(* IEC 61131-3 sources: TIA2AX/tests/test_projects/expected/HW_2200220OffsetBodu_V18/A5, 6 files *)

(* ---- HwInputs.st ---- *)
TYPE
	HwInputs : STRUCT
		A6_15A2 AT %B0 : WORD;
		A6_15A3 AT %B2 : WORD;
		A6_15A4 AT %B4 : WORD;
		A6_15A9 AT %B6 : ARRAY[0..7] OF BYTE;
		_52K1_53AB1 AT %B157 : BYTE;
		_52K1_54AB2 AT %B158 : BYTE;
		_52K1_55AB3 AT %B159 : BYTE;
		_52K1_56AB4 AT %B160 : BYTE;
		_52K1_57AB5 AT %B179 : BYTE;
		_52K1_58AB6 AT %B147 : ARRAY[0..7] OF BYTE;
		_52K1_59AB7 AT %B45 : BYTE;
		_52K1_59aAB7 AT %B155 : BYTE;
		_52K1_60AB8 AT %B156 : BYTE;
		_52K1_61AB9 AT %B161 : BYTE;
		_52K1_62AB10 AT %B178 : BYTE;
		Bash_Input_1_byte_1 AT %B5300 : BYTE;
		Bash_Input_1_byte_2 AT %B5301 : BYTE;
		Bash_Input_2_word_1 AT %B5302 : DWORD;
		Bash_Input_1_word_1 AT %B5306 : WORD;
		Bash_Input_2_word_2 AT %B5308 : DWORD;
		Bash_Input_1_word_2 AT %B5312 : WORD;
		AEBDown_Input_1_byte_1 AT %B5314 : BYTE;
		AEBDown_Input_1_byte_2 AT %B5315 : BYTE;
		AEBDown_Input_2_word_1 AT %B5316 : DWORD;
		AEBDown_Input_1_word_1 AT %B5320 : WORD;
		AEBDown_Input_2_word_2 AT %B5322 : DWORD;
		AEBDown_Input_1_word_2 AT %B5326 : WORD;
		AEBUp_Input_1_byte_1 AT %B5328 : BYTE;
		AEBUp_Input_1_byte_2 AT %B5329 : BYTE;
		AEBUp_Input_2_word_1 AT %B5330 : DWORD;
		AEBUp_Input_1_word_1 AT %B5334 : WORD;
		AEBUp_Input_2_word_2 AT %B5336 : DWORD;
		AEBUp_Input_1_word_2 AT %B5340 : WORD;
		AETDown_Input_1_byte_1 AT %B5342 : BYTE;
		AETDown_Input_1_byte_2 AT %B5343 : BYTE;
		AETDown_Input_2_word_1 AT %B5344 : DWORD;
		AETDown_Input_1_word_1 AT %B5348 : WORD;
		AETDown_Input_2_word_2 AT %B5350 : DWORD;
		AETDown_Input_1_word_2 AT %B5354 : WORD;
		AETUp_Input_1_byte_1 AT %B5356 : BYTE;
		AETUp_Input_1_byte_2 AT %B5357 : BYTE;
		AETUp_Input_2_word_1 AT %B5358 : DWORD;
		AETUp_Input_1_word_1 AT %B5362 : WORD;
		AETUp_Input_2_word_2 AT %B5364 : DWORD;
		AETUp_Input_1_word_2 AT %B5368 : WORD;
		GT2_DL_PN1_1 AT %B162 : ARRAY[0..15] OF BYTE;
		GT2_B1 AT %B228 : ARRAY[0..6] OF BYTE;
		GT2_B2 AT %B221 : ARRAY[0..6] OF BYTE;
		GT2_B3 AT %B214 : ARRAY[0..6] OF BYTE;
		GT2_B4 AT %B207 : ARRAY[0..6] OF BYTE;
		GT2_B5 AT %B200 : ARRAY[0..6] OF BYTE;
		GT2_B6 AT %B189 : ARRAY[0..6] OF BYTE;
		GT2_B7 AT %B182 : ARRAY[0..6] OF BYTE;
		GT2_B8 AT %B235 : ARRAY[0..6] OF BYTE;
		GT2_B9 AT %B242 : ARRAY[0..6] OF BYTE;
		CPX_CW_SW AT %B71 : DWORD;
		CPX_CNC AT %B408 : ARRAY[0..31] OF BYTE;
		CPX_PtP AT %B385 : ARRAY[0..15] OF BYTE;
		CPX_Error AT %B440 : ARRAY[0..31] OF BYTE;
		Reader_Handshake_and_General_Error_Status_Bits_1 AT %B15 : BYTE;
		Reader_BUSY_Status_Bits_1 AT %B16 : BYTE;
		Reader_Completion_Status_Bits_1 AT %B17 : BYTE;
		Reader_Error_Status_Bits_1 AT %B18 : BYTE;
		Reader_Terminal_Status_Bits_1 AT %B19 : BYTE;
		Reader_Unstable_Read_Status_Bits_1 AT %B20 : BYTE;
		Reader_Matching_Level_and_Total_Evaluation_Grade_Status_1 AT %B21 : ARRAY[0..7] OF BYTE;
		Reader_Operation_Result_Status_1 AT %B51 : ARRAY[0..19] OF BYTE;
		Reader_Read_Data_128Byte_1 AT %B249 : ARRAY[0..135] OF BYTE;
	END_STRUCT;
END_TYPE

(* ---- HwOutputs.st ---- *)
TYPE
	HwOutputs : STRUCT
		A6_15A5 AT %B1 : WORD;
		A6_15A6 AT %B3 : WORD;
		A6_15A7 AT %B14 : WORD;
		A6_15A8 AT %B16 : WORD;
		A6_15A10 AT %B99 : ARRAY[0..7] OF BYTE;
		VI_13_MPA1S_VMPA1_FB_EMS_8_8DO_1 AT %B6 : BYTE;
		VI_13_MPA1S_VMPA1_FB_EMS_8_8DO_2 AT %B8 : BYTE;
		VI_13_MPA1S_VMPA1_FB_EMS_8_8DO_3 AT %B9 : BYTE;
		VI_13_MPA1S_VMPA1_FB_EMS_8_8DO_4 AT %B10 : BYTE;
		VI_13_MPA1S_VMPA1_FB_EMS_8_8DO_5 AT %B11 : BYTE;
		VI_13_MPA1S_VMPA1_FB_EMS_8_8DO_6 AT %B12 : BYTE;
		VI_13_MPA1S_VMPA1_FB_EMS_8_8DO_7 AT %B13 : BYTE;
		VI_13_MPA1S_VMPA1_FB_EMS_8_8DO_8 AT %B18 : BYTE;
		Bash_Output_1_byte_1 AT %B5300 : BYTE;
		Bash_Output_1_byte_2 AT %B5301 : BYTE;
		AEBDown_Output_1_byte_1 AT %B5302 : BYTE;
		AEBDown_Output_1_byte_2 AT %B5303 : BYTE;
		AEBUp_Output_1_byte_1 AT %B5304 : BYTE;
		AEBUp_Output_1_byte_2 AT %B5305 : BYTE;
		AETDown_Output_1_byte_1 AT %B5306 : BYTE;
		AETDown_Output_1_byte_2 AT %B5307 : BYTE;
		AETUp_Output_1_byte_1 AT %B5308 : BYTE;
		AETUp_Output_1_byte_2 AT %B5309 : BYTE;
		GT2_DL_PN1_1 AT %B32 : BYTE;
		GT2_B1 AT %B45 : BYTE;
		GT2_B2 AT %B147 : BYTE;
		GT2_B3 AT %B148 : BYTE;
		GT2_B4 AT %B149 : BYTE;
		GT2_B5 AT %B39 : BYTE;
		GT2_B6 AT %B38 : BYTE;
		GT2_B7 AT %B150 : BYTE;
		GT2_B8 AT %B151 : BYTE;
		GT2_B9 AT %B33 : BYTE;
		CPX_CW_SW AT %B21 : DWORD;
		CPX_CNC AT %B51 : ARRAY[0..31] OF BYTE;
		CPX_PtP AT %B83 : ARRAY[0..15] OF BYTE;
		CPX_Error AT %B282 : ARRAY[0..31] OF BYTE;
		Reader_Latch_and_Error_Clear_Control_Bits_1 AT %B0 : BYTE;
		Reader_Operation_instruction_Control_Bits_1 AT %B5 : BYTE;
		Reader_Completion_Clear_Control_Bits_1 AT %B7 : BYTE;
		Reader_Parameter_Bank_Number_1 AT %B19 : WORD;
		Reader_User_Data_128Byte_1 AT %B152 : ARRAY[0..129] OF BYTE;
	END_STRUCT;
END_TYPE

(* ---- PlcInputs.st ---- *)
TYPE
	PlcInputs : STRUCT
		A6_15A2 : WORD;
		A6_15A3 : WORD;
		A6_15A4 : WORD;
		A6_15A9 : ARRAY[0..7] OF BYTE;
		_52K1_53AB1 : BYTE;
		_52K1_54AB2 : BYTE;
		_52K1_55AB3 : BYTE;
		_52K1_56AB4 : BYTE;
		_52K1_57AB5 : BYTE;
		_52K1_58AB6 : ARRAY[0..7] OF BYTE;
		_52K1_59AB7 : BYTE;
		_52K1_59aAB7 : BYTE;
		_52K1_60AB8 : BYTE;
		_52K1_61AB9 : BYTE;
		_52K1_62AB10 : BYTE;
		Bash_Input_1_byte_1 : BYTE;
		Bash_Input_1_byte_2 : BYTE;
		Bash_Input_2_word_1 : DWORD;
		Bash_Input_1_word_1 : WORD;
		Bash_Input_2_word_2 : DWORD;
		Bash_Input_1_word_2 : WORD;
		AEBDown_Input_1_byte_1 : BYTE;
		AEBDown_Input_1_byte_2 : BYTE;
		AEBDown_Input_2_word_1 : DWORD;
		AEBDown_Input_1_word_1 : WORD;
		AEBDown_Input_2_word_2 : DWORD;
		AEBDown_Input_1_word_2 : WORD;
		AEBUp_Input_1_byte_1 : BYTE;
		AEBUp_Input_1_byte_2 : BYTE;
		AEBUp_Input_2_word_1 : DWORD;
		AEBUp_Input_1_word_1 : WORD;
		AEBUp_Input_2_word_2 : DWORD;
		AEBUp_Input_1_word_2 : WORD;
		AETDown_Input_1_byte_1 : BYTE;
		AETDown_Input_1_byte_2 : BYTE;
		AETDown_Input_2_word_1 : DWORD;
		AETDown_Input_1_word_1 : WORD;
		AETDown_Input_2_word_2 : DWORD;
		AETDown_Input_1_word_2 : WORD;
		AETUp_Input_1_byte_1 : BYTE;
		AETUp_Input_1_byte_2 : BYTE;
		AETUp_Input_2_word_1 : DWORD;
		AETUp_Input_1_word_1 : WORD;
		AETUp_Input_2_word_2 : DWORD;
		AETUp_Input_1_word_2 : WORD;
		GT2_DL_PN1_1 : ARRAY[0..15] OF BYTE;
		GT2_B1 : ARRAY[0..6] OF BYTE;
		GT2_B2 : ARRAY[0..6] OF BYTE;
		GT2_B3 : ARRAY[0..6] OF BYTE;
		GT2_B4 : ARRAY[0..6] OF BYTE;
		GT2_B5 : ARRAY[0..6] OF BYTE;
		GT2_B6 : ARRAY[0..6] OF BYTE;
		GT2_B7 : ARRAY[0..6] OF BYTE;
		GT2_B8 : ARRAY[0..6] OF BYTE;
		GT2_B9 : ARRAY[0..6] OF BYTE;
		CPX_CW_SW : DWORD;
		CPX_CNC : ARRAY[0..31] OF BYTE;
		CPX_PtP : ARRAY[0..15] OF BYTE;
		CPX_Error : ARRAY[0..31] OF BYTE;
		Reader_Handshake_and_General_Error_Status_Bits_1 : BYTE;
		Reader_BUSY_Status_Bits_1 : BYTE;
		Reader_Completion_Status_Bits_1 : BYTE;
		Reader_Error_Status_Bits_1 : BYTE;
		Reader_Terminal_Status_Bits_1 : BYTE;
		Reader_Unstable_Read_Status_Bits_1 : BYTE;
		Reader_Matching_Level_and_Total_Evaluation_Grade_Status_1 : ARRAY[0..7] OF BYTE;
		Reader_Operation_Result_Status_1 : ARRAY[0..19] OF BYTE;
		Reader_Read_Data_128Byte_1 : ARRAY[0..135] OF BYTE;
	END_STRUCT;
END_TYPE

(* ---- PlcOutputs.st ---- *)
TYPE
	PlcOutputs : STRUCT
		A6_15A5 : WORD;
		A6_15A6 : WORD;
		A6_15A7 : WORD;
		A6_15A8 : WORD;
		A6_15A10 : ARRAY[0..7] OF BYTE;
		VI_13_MPA1S_VMPA1_FB_EMS_8_8DO_1 : BYTE;
		VI_13_MPA1S_VMPA1_FB_EMS_8_8DO_2 : BYTE;
		VI_13_MPA1S_VMPA1_FB_EMS_8_8DO_3 : BYTE;
		VI_13_MPA1S_VMPA1_FB_EMS_8_8DO_4 : BYTE;
		VI_13_MPA1S_VMPA1_FB_EMS_8_8DO_5 : BYTE;
		VI_13_MPA1S_VMPA1_FB_EMS_8_8DO_6 : BYTE;
		VI_13_MPA1S_VMPA1_FB_EMS_8_8DO_7 : BYTE;
		VI_13_MPA1S_VMPA1_FB_EMS_8_8DO_8 : BYTE;
		Bash_Output_1_byte_1 : BYTE;
		Bash_Output_1_byte_2 : BYTE;
		AEBDown_Output_1_byte_1 : BYTE;
		AEBDown_Output_1_byte_2 : BYTE;
		AEBUp_Output_1_byte_1 : BYTE;
		AEBUp_Output_1_byte_2 : BYTE;
		AETDown_Output_1_byte_1 : BYTE;
		AETDown_Output_1_byte_2 : BYTE;
		AETUp_Output_1_byte_1 : BYTE;
		AETUp_Output_1_byte_2 : BYTE;
		GT2_DL_PN1_1 : BYTE;
		GT2_B1 : BYTE;
		GT2_B2 : BYTE;
		GT2_B3 : BYTE;
		GT2_B4 : BYTE;
		GT2_B5 : BYTE;
		GT2_B6 : BYTE;
		GT2_B7 : BYTE;
		GT2_B8 : BYTE;
		GT2_B9 : BYTE;
		CPX_CW_SW : DWORD;
		CPX_CNC : ARRAY[0..31] OF BYTE;
		CPX_PtP : ARRAY[0..15] OF BYTE;
		CPX_Error : ARRAY[0..31] OF BYTE;
		Reader_Latch_and_Error_Clear_Control_Bits_1 : BYTE;
		Reader_Operation_instruction_Control_Bits_1 : BYTE;
		Reader_Completion_Clear_Control_Bits_1 : BYTE;
		Reader_Parameter_Bank_Number_1 : WORD;
		Reader_User_Data_128Byte_1 : ARRAY[0..129] OF BYTE;
	END_STRUCT;
END_TYPE

(* ---- CopyInputs.st ---- *)
FUNCTION CopyInputs
	VAR_EXTERNAL
		HwInputs : HwInputs;
		PlcInputs : PlcInputs;
	END_VAR
	PlcInputs.A6_15A2 := HwInputs.A6_15A2;
	PlcInputs.A6_15A3 := HwInputs.A6_15A3;
	PlcInputs.A6_15A4 := HwInputs.A6_15A4;
	PlcInputs.A6_15A9[0] := HwInputs.A6_15A9[0];
	PlcInputs.A6_15A9[1] := HwInputs.A6_15A9[1];
	PlcInputs.A6_15A9[2] := HwInputs.A6_15A9[2];
	PlcInputs.A6_15A9[3] := HwInputs.A6_15A9[3];
	PlcInputs.A6_15A9[4] := HwInputs.A6_15A9[4];
	PlcInputs.A6_15A9[5] := HwInputs.A6_15A9[5];
	PlcInputs.A6_15A9[6] := HwInputs.A6_15A9[6];
	PlcInputs.A6_15A9[7] := HwInputs.A6_15A9[7];
	PlcInputs._52K1_53AB1 := HwInputs._52K1_53AB1;
	PlcInputs._52K1_54AB2 := HwInputs._52K1_54AB2;
	PlcInputs._52K1_55AB3 := HwInputs._52K1_55AB3;
	PlcInputs._52K1_56AB4 := HwInputs._52K1_56AB4;
	PlcInputs._52K1_57AB5 := HwInputs._52K1_57AB5;
	PlcInputs._52K1_58AB6[0] := HwInputs._52K1_58AB6[0];
	PlcInputs._52K1_58AB6[1] := HwInputs._52K1_58AB6[1];
	PlcInputs._52K1_58AB6[2] := HwInputs._52K1_58AB6[2];
	PlcInputs._52K1_58AB6[3] := HwInputs._52K1_58AB6[3];
	PlcInputs._52K1_58AB6[4] := HwInputs._52K1_58AB6[4];
	PlcInputs._52K1_58AB6[5] := HwInputs._52K1_58AB6[5];
	PlcInputs._52K1_58AB6[6] := HwInputs._52K1_58AB6[6];
	PlcInputs._52K1_58AB6[7] := HwInputs._52K1_58AB6[7];
	PlcInputs._52K1_59AB7 := HwInputs._52K1_59AB7;
	PlcInputs._52K1_59aAB7 := HwInputs._52K1_59aAB7;
	PlcInputs._52K1_60AB8 := HwInputs._52K1_60AB8;
	PlcInputs._52K1_61AB9 := HwInputs._52K1_61AB9;
	PlcInputs._52K1_62AB10 := HwInputs._52K1_62AB10;
	PlcInputs.Bash_Input_1_byte_1 := HwInputs.Bash_Input_1_byte_1;
	PlcInputs.Bash_Input_1_byte_2 := HwInputs.Bash_Input_1_byte_2;
	PlcInputs.Bash_Input_2_word_1 := HwInputs.Bash_Input_2_word_1;
	PlcInputs.Bash_Input_1_word_1 := HwInputs.Bash_Input_1_word_1;
	PlcInputs.Bash_Input_2_word_2 := HwInputs.Bash_Input_2_word_2;
	PlcInputs.Bash_Input_1_word_2 := HwInputs.Bash_Input_1_word_2;
	PlcInputs.AEBDown_Input_1_byte_1 := HwInputs.AEBDown_Input_1_byte_1;
	PlcInputs.AEBDown_Input_1_byte_2 := HwInputs.AEBDown_Input_1_byte_2;
	PlcInputs.AEBDown_Input_2_word_1 := HwInputs.AEBDown_Input_2_word_1;
	PlcInputs.AEBDown_Input_1_word_1 := HwInputs.AEBDown_Input_1_word_1;
	PlcInputs.AEBDown_Input_2_word_2 := HwInputs.AEBDown_Input_2_word_2;
	PlcInputs.AEBDown_Input_1_word_2 := HwInputs.AEBDown_Input_1_word_2;
	PlcInputs.AEBUp_Input_1_byte_1 := HwInputs.AEBUp_Input_1_byte_1;
	PlcInputs.AEBUp_Input_1_byte_2 := HwInputs.AEBUp_Input_1_byte_2;
	PlcInputs.AEBUp_Input_2_word_1 := HwInputs.AEBUp_Input_2_word_1;
	PlcInputs.AEBUp_Input_1_word_1 := HwInputs.AEBUp_Input_1_word_1;
	PlcInputs.AEBUp_Input_2_word_2 := HwInputs.AEBUp_Input_2_word_2;
	PlcInputs.AEBUp_Input_1_word_2 := HwInputs.AEBUp_Input_1_word_2;
	PlcInputs.AETDown_Input_1_byte_1 := HwInputs.AETDown_Input_1_byte_1;
	PlcInputs.AETDown_Input_1_byte_2 := HwInputs.AETDown_Input_1_byte_2;
	PlcInputs.AETDown_Input_2_word_1 := HwInputs.AETDown_Input_2_word_1;
	PlcInputs.AETDown_Input_1_word_1 := HwInputs.AETDown_Input_1_word_1;
	PlcInputs.AETDown_Input_2_word_2 := HwInputs.AETDown_Input_2_word_2;
	PlcInputs.AETDown_Input_1_word_2 := HwInputs.AETDown_Input_1_word_2;
	PlcInputs.AETUp_Input_1_byte_1 := HwInputs.AETUp_Input_1_byte_1;
	PlcInputs.AETUp_Input_1_byte_2 := HwInputs.AETUp_Input_1_byte_2;
	PlcInputs.AETUp_Input_2_word_1 := HwInputs.AETUp_Input_2_word_1;
	PlcInputs.AETUp_Input_1_word_1 := HwInputs.AETUp_Input_1_word_1;
	PlcInputs.AETUp_Input_2_word_2 := HwInputs.AETUp_Input_2_word_2;
	PlcInputs.AETUp_Input_1_word_2 := HwInputs.AETUp_Input_1_word_2;
	PlcInputs.GT2_DL_PN1_1[0] := HwInputs.GT2_DL_PN1_1[0];
	PlcInputs.GT2_DL_PN1_1[1] := HwInputs.GT2_DL_PN1_1[1];
	PlcInputs.GT2_DL_PN1_1[2] := HwInputs.GT2_DL_PN1_1[2];
	PlcInputs.GT2_DL_PN1_1[3] := HwInputs.GT2_DL_PN1_1[3];
	PlcInputs.GT2_DL_PN1_1[4] := HwInputs.GT2_DL_PN1_1[4];
	PlcInputs.GT2_DL_PN1_1[5] := HwInputs.GT2_DL_PN1_1[5];
	PlcInputs.GT2_DL_PN1_1[6] := HwInputs.GT2_DL_PN1_1[6];
	PlcInputs.GT2_DL_PN1_1[7] := HwInputs.GT2_DL_PN1_1[7];
	PlcInputs.GT2_DL_PN1_1[8] := HwInputs.GT2_DL_PN1_1[8];
	PlcInputs.GT2_DL_PN1_1[9] := HwInputs.GT2_DL_PN1_1[9];
	PlcInputs.GT2_DL_PN1_1[10] := HwInputs.GT2_DL_PN1_1[10];
	PlcInputs.GT2_DL_PN1_1[11] := HwInputs.GT2_DL_PN1_1[11];
	PlcInputs.GT2_DL_PN1_1[12] := HwInputs.GT2_DL_PN1_1[12];
	PlcInputs.GT2_DL_PN1_1[13] := HwInputs.GT2_DL_PN1_1[13];
	PlcInputs.GT2_DL_PN1_1[14] := HwInputs.GT2_DL_PN1_1[14];
	PlcInputs.GT2_DL_PN1_1[15] := HwInputs.GT2_DL_PN1_1[15];
	PlcInputs.GT2_B1[0] := HwInputs.GT2_B1[0];
	PlcInputs.GT2_B1[1] := HwInputs.GT2_B1[1];
	PlcInputs.GT2_B1[2] := HwInputs.GT2_B1[2];
	PlcInputs.GT2_B1[3] := HwInputs.GT2_B1[3];
	PlcInputs.GT2_B1[4] := HwInputs.GT2_B1[4];
	PlcInputs.GT2_B1[5] := HwInputs.GT2_B1[5];
	PlcInputs.GT2_B1[6] := HwInputs.GT2_B1[6];
	PlcInputs.GT2_B2[0] := HwInputs.GT2_B2[0];
	PlcInputs.GT2_B2[1] := HwInputs.GT2_B2[1];
	PlcInputs.GT2_B2[2] := HwInputs.GT2_B2[2];
	PlcInputs.GT2_B2[3] := HwInputs.GT2_B2[3];
	PlcInputs.GT2_B2[4] := HwInputs.GT2_B2[4];
	PlcInputs.GT2_B2[5] := HwInputs.GT2_B2[5];
	PlcInputs.GT2_B2[6] := HwInputs.GT2_B2[6];
	PlcInputs.GT2_B3[0] := HwInputs.GT2_B3[0];
	PlcInputs.GT2_B3[1] := HwInputs.GT2_B3[1];
	PlcInputs.GT2_B3[2] := HwInputs.GT2_B3[2];
	PlcInputs.GT2_B3[3] := HwInputs.GT2_B3[3];
	PlcInputs.GT2_B3[4] := HwInputs.GT2_B3[4];
	PlcInputs.GT2_B3[5] := HwInputs.GT2_B3[5];
	PlcInputs.GT2_B3[6] := HwInputs.GT2_B3[6];
	PlcInputs.GT2_B4[0] := HwInputs.GT2_B4[0];
	PlcInputs.GT2_B4[1] := HwInputs.GT2_B4[1];
	PlcInputs.GT2_B4[2] := HwInputs.GT2_B4[2];
	PlcInputs.GT2_B4[3] := HwInputs.GT2_B4[3];
	PlcInputs.GT2_B4[4] := HwInputs.GT2_B4[4];
	PlcInputs.GT2_B4[5] := HwInputs.GT2_B4[5];
	PlcInputs.GT2_B4[6] := HwInputs.GT2_B4[6];
	PlcInputs.GT2_B5[0] := HwInputs.GT2_B5[0];
	PlcInputs.GT2_B5[1] := HwInputs.GT2_B5[1];
	PlcInputs.GT2_B5[2] := HwInputs.GT2_B5[2];
	PlcInputs.GT2_B5[3] := HwInputs.GT2_B5[3];
	PlcInputs.GT2_B5[4] := HwInputs.GT2_B5[4];
	PlcInputs.GT2_B5[5] := HwInputs.GT2_B5[5];
	PlcInputs.GT2_B5[6] := HwInputs.GT2_B5[6];
	PlcInputs.GT2_B6[0] := HwInputs.GT2_B6[0];
	PlcInputs.GT2_B6[1] := HwInputs.GT2_B6[1];
	PlcInputs.GT2_B6[2] := HwInputs.GT2_B6[2];
	PlcInputs.GT2_B6[3] := HwInputs.GT2_B6[3];
	PlcInputs.GT2_B6[4] := HwInputs.GT2_B6[4];
	PlcInputs.GT2_B6[5] := HwInputs.GT2_B6[5];
	PlcInputs.GT2_B6[6] := HwInputs.GT2_B6[6];
	PlcInputs.GT2_B7[0] := HwInputs.GT2_B7[0];
	PlcInputs.GT2_B7[1] := HwInputs.GT2_B7[1];
	PlcInputs.GT2_B7[2] := HwInputs.GT2_B7[2];
	PlcInputs.GT2_B7[3] := HwInputs.GT2_B7[3];
	PlcInputs.GT2_B7[4] := HwInputs.GT2_B7[4];
	PlcInputs.GT2_B7[5] := HwInputs.GT2_B7[5];
	PlcInputs.GT2_B7[6] := HwInputs.GT2_B7[6];
	PlcInputs.GT2_B8[0] := HwInputs.GT2_B8[0];
	PlcInputs.GT2_B8[1] := HwInputs.GT2_B8[1];
	PlcInputs.GT2_B8[2] := HwInputs.GT2_B8[2];
	PlcInputs.GT2_B8[3] := HwInputs.GT2_B8[3];
	PlcInputs.GT2_B8[4] := HwInputs.GT2_B8[4];
	PlcInputs.GT2_B8[5] := HwInputs.GT2_B8[5];
	PlcInputs.GT2_B8[6] := HwInputs.GT2_B8[6];
	PlcInputs.GT2_B9[0] := HwInputs.GT2_B9[0];
	PlcInputs.GT2_B9[1] := HwInputs.GT2_B9[1];
	PlcInputs.GT2_B9[2] := HwInputs.GT2_B9[2];
	PlcInputs.GT2_B9[3] := HwInputs.GT2_B9[3];
	PlcInputs.GT2_B9[4] := HwInputs.GT2_B9[4];
	PlcInputs.GT2_B9[5] := HwInputs.GT2_B9[5];
	PlcInputs.GT2_B9[6] := HwInputs.GT2_B9[6];
	PlcInputs.CPX_CW_SW := HwInputs.CPX_CW_SW;
	PlcInputs.CPX_CNC[0] := HwInputs.CPX_CNC[0];
	PlcInputs.CPX_CNC[1] := HwInputs.CPX_CNC[1];
	PlcInputs.CPX_CNC[2] := HwInputs.CPX_CNC[2];
	PlcInputs.CPX_CNC[3] := HwInputs.CPX_CNC[3];
	PlcInputs.CPX_CNC[4] := HwInputs.CPX_CNC[4];
	PlcInputs.CPX_CNC[5] := HwInputs.CPX_CNC[5];
	PlcInputs.CPX_CNC[6] := HwInputs.CPX_CNC[6];
	PlcInputs.CPX_CNC[7] := HwInputs.CPX_CNC[7];
	PlcInputs.CPX_CNC[8] := HwInputs.CPX_CNC[8];
	PlcInputs.CPX_CNC[9] := HwInputs.CPX_CNC[9];
	PlcInputs.CPX_CNC[10] := HwInputs.CPX_CNC[10];
	PlcInputs.CPX_CNC[11] := HwInputs.CPX_CNC[11];
	PlcInputs.CPX_CNC[12] := HwInputs.CPX_CNC[12];
	PlcInputs.CPX_CNC[13] := HwInputs.CPX_CNC[13];
	PlcInputs.CPX_CNC[14] := HwInputs.CPX_CNC[14];
	PlcInputs.CPX_CNC[15] := HwInputs.CPX_CNC[15];
	PlcInputs.CPX_CNC[16] := HwInputs.CPX_CNC[16];
	PlcInputs.CPX_CNC[17] := HwInputs.CPX_CNC[17];
	PlcInputs.CPX_CNC[18] := HwInputs.CPX_CNC[18];
	PlcInputs.CPX_CNC[19] := HwInputs.CPX_CNC[19];
	PlcInputs.CPX_CNC[20] := HwInputs.CPX_CNC[20];
	PlcInputs.CPX_CNC[21] := HwInputs.CPX_CNC[21];
	PlcInputs.CPX_CNC[22] := HwInputs.CPX_CNC[22];
	PlcInputs.CPX_CNC[23] := HwInputs.CPX_CNC[23];
	PlcInputs.CPX_CNC[24] := HwInputs.CPX_CNC[24];
	PlcInputs.CPX_CNC[25] := HwInputs.CPX_CNC[25];
	PlcInputs.CPX_CNC[26] := HwInputs.CPX_CNC[26];
	PlcInputs.CPX_CNC[27] := HwInputs.CPX_CNC[27];
	PlcInputs.CPX_CNC[28] := HwInputs.CPX_CNC[28];
	PlcInputs.CPX_CNC[29] := HwInputs.CPX_CNC[29];
	PlcInputs.CPX_CNC[30] := HwInputs.CPX_CNC[30];
	PlcInputs.CPX_CNC[31] := HwInputs.CPX_CNC[31];
	PlcInputs.CPX_PtP[0] := HwInputs.CPX_PtP[0];
	PlcInputs.CPX_PtP[1] := HwInputs.CPX_PtP[1];
	PlcInputs.CPX_PtP[2] := HwInputs.CPX_PtP[2];
	PlcInputs.CPX_PtP[3] := HwInputs.CPX_PtP[3];
	PlcInputs.CPX_PtP[4] := HwInputs.CPX_PtP[4];
	PlcInputs.CPX_PtP[5] := HwInputs.CPX_PtP[5];
	PlcInputs.CPX_PtP[6] := HwInputs.CPX_PtP[6];
	PlcInputs.CPX_PtP[7] := HwInputs.CPX_PtP[7];
	PlcInputs.CPX_PtP[8] := HwInputs.CPX_PtP[8];
	PlcInputs.CPX_PtP[9] := HwInputs.CPX_PtP[9];
	PlcInputs.CPX_PtP[10] := HwInputs.CPX_PtP[10];
	PlcInputs.CPX_PtP[11] := HwInputs.CPX_PtP[11];
	PlcInputs.CPX_PtP[12] := HwInputs.CPX_PtP[12];
	PlcInputs.CPX_PtP[13] := HwInputs.CPX_PtP[13];
	PlcInputs.CPX_PtP[14] := HwInputs.CPX_PtP[14];
	PlcInputs.CPX_PtP[15] := HwInputs.CPX_PtP[15];
	PlcInputs.CPX_Error[0] := HwInputs.CPX_Error[0];
	PlcInputs.CPX_Error[1] := HwInputs.CPX_Error[1];
	PlcInputs.CPX_Error[2] := HwInputs.CPX_Error[2];
	PlcInputs.CPX_Error[3] := HwInputs.CPX_Error[3];
	PlcInputs.CPX_Error[4] := HwInputs.CPX_Error[4];
	PlcInputs.CPX_Error[5] := HwInputs.CPX_Error[5];
	PlcInputs.CPX_Error[6] := HwInputs.CPX_Error[6];
	PlcInputs.CPX_Error[7] := HwInputs.CPX_Error[7];
	PlcInputs.CPX_Error[8] := HwInputs.CPX_Error[8];
	PlcInputs.CPX_Error[9] := HwInputs.CPX_Error[9];
	PlcInputs.CPX_Error[10] := HwInputs.CPX_Error[10];
	PlcInputs.CPX_Error[11] := HwInputs.CPX_Error[11];
	PlcInputs.CPX_Error[12] := HwInputs.CPX_Error[12];
	PlcInputs.CPX_Error[13] := HwInputs.CPX_Error[13];
	PlcInputs.CPX_Error[14] := HwInputs.CPX_Error[14];
	PlcInputs.CPX_Error[15] := HwInputs.CPX_Error[15];
	PlcInputs.CPX_Error[16] := HwInputs.CPX_Error[16];
	PlcInputs.CPX_Error[17] := HwInputs.CPX_Error[17];
	PlcInputs.CPX_Error[18] := HwInputs.CPX_Error[18];
	PlcInputs.CPX_Error[19] := HwInputs.CPX_Error[19];
	PlcInputs.CPX_Error[20] := HwInputs.CPX_Error[20];
	PlcInputs.CPX_Error[21] := HwInputs.CPX_Error[21];
	PlcInputs.CPX_Error[22] := HwInputs.CPX_Error[22];
	PlcInputs.CPX_Error[23] := HwInputs.CPX_Error[23];
	PlcInputs.CPX_Error[24] := HwInputs.CPX_Error[24];
	PlcInputs.CPX_Error[25] := HwInputs.CPX_Error[25];
	PlcInputs.CPX_Error[26] := HwInputs.CPX_Error[26];
	PlcInputs.CPX_Error[27] := HwInputs.CPX_Error[27];
	PlcInputs.CPX_Error[28] := HwInputs.CPX_Error[28];
	PlcInputs.CPX_Error[29] := HwInputs.CPX_Error[29];
	PlcInputs.CPX_Error[30] := HwInputs.CPX_Error[30];
	PlcInputs.CPX_Error[31] := HwInputs.CPX_Error[31];
	PlcInputs.Reader_Handshake_and_General_Error_Status_Bits_1 := HwInputs.Reader_Handshake_and_General_Error_Status_Bits_1;
	PlcInputs.Reader_BUSY_Status_Bits_1 := HwInputs.Reader_BUSY_Status_Bits_1;
	PlcInputs.Reader_Completion_Status_Bits_1 := HwInputs.Reader_Completion_Status_Bits_1;
	PlcInputs.Reader_Error_Status_Bits_1 := HwInputs.Reader_Error_Status_Bits_1;
	PlcInputs.Reader_Terminal_Status_Bits_1 := HwInputs.Reader_Terminal_Status_Bits_1;
	PlcInputs.Reader_Unstable_Read_Status_Bits_1 := HwInputs.Reader_Unstable_Read_Status_Bits_1;
	PlcInputs.Reader_Matching_Level_and_Total_Evaluation_Grade_Status_1[0] := HwInputs.Reader_Matching_Level_and_Total_Evaluation_Grade_Status_1[0];
	PlcInputs.Reader_Matching_Level_and_Total_Evaluation_Grade_Status_1[1] := HwInputs.Reader_Matching_Level_and_Total_Evaluation_Grade_Status_1[1];
	PlcInputs.Reader_Matching_Level_and_Total_Evaluation_Grade_Status_1[2] := HwInputs.Reader_Matching_Level_and_Total_Evaluation_Grade_Status_1[2];
	PlcInputs.Reader_Matching_Level_and_Total_Evaluation_Grade_Status_1[3] := HwInputs.Reader_Matching_Level_and_Total_Evaluation_Grade_Status_1[3];
	PlcInputs.Reader_Matching_Level_and_Total_Evaluation_Grade_Status_1[4] := HwInputs.Reader_Matching_Level_and_Total_Evaluation_Grade_Status_1[4];
	PlcInputs.Reader_Matching_Level_and_Total_Evaluation_Grade_Status_1[5] := HwInputs.Reader_Matching_Level_and_Total_Evaluation_Grade_Status_1[5];
	PlcInputs.Reader_Matching_Level_and_Total_Evaluation_Grade_Status_1[6] := HwInputs.Reader_Matching_Level_and_Total_Evaluation_Grade_Status_1[6];
	PlcInputs.Reader_Matching_Level_and_Total_Evaluation_Grade_Status_1[7] := HwInputs.Reader_Matching_Level_and_Total_Evaluation_Grade_Status_1[7];
	PlcInputs.Reader_Operation_Result_Status_1[0] := HwInputs.Reader_Operation_Result_Status_1[0];
	PlcInputs.Reader_Operation_Result_Status_1[1] := HwInputs.Reader_Operation_Result_Status_1[1];
	PlcInputs.Reader_Operation_Result_Status_1[2] := HwInputs.Reader_Operation_Result_Status_1[2];
	PlcInputs.Reader_Operation_Result_Status_1[3] := HwInputs.Reader_Operation_Result_Status_1[3];
	PlcInputs.Reader_Operation_Result_Status_1[4] := HwInputs.Reader_Operation_Result_Status_1[4];
	PlcInputs.Reader_Operation_Result_Status_1[5] := HwInputs.Reader_Operation_Result_Status_1[5];
	PlcInputs.Reader_Operation_Result_Status_1[6] := HwInputs.Reader_Operation_Result_Status_1[6];
	PlcInputs.Reader_Operation_Result_Status_1[7] := HwInputs.Reader_Operation_Result_Status_1[7];
	PlcInputs.Reader_Operation_Result_Status_1[8] := HwInputs.Reader_Operation_Result_Status_1[8];
	PlcInputs.Reader_Operation_Result_Status_1[9] := HwInputs.Reader_Operation_Result_Status_1[9];
	PlcInputs.Reader_Operation_Result_Status_1[10] := HwInputs.Reader_Operation_Result_Status_1[10];
	PlcInputs.Reader_Operation_Result_Status_1[11] := HwInputs.Reader_Operation_Result_Status_1[11];
	PlcInputs.Reader_Operation_Result_Status_1[12] := HwInputs.Reader_Operation_Result_Status_1[12];
	PlcInputs.Reader_Operation_Result_Status_1[13] := HwInputs.Reader_Operation_Result_Status_1[13];
	PlcInputs.Reader_Operation_Result_Status_1[14] := HwInputs.Reader_Operation_Result_Status_1[14];
	PlcInputs.Reader_Operation_Result_Status_1[15] := HwInputs.Reader_Operation_Result_Status_1[15];
	PlcInputs.Reader_Operation_Result_Status_1[16] := HwInputs.Reader_Operation_Result_Status_1[16];
	PlcInputs.Reader_Operation_Result_Status_1[17] := HwInputs.Reader_Operation_Result_Status_1[17];
	PlcInputs.Reader_Operation_Result_Status_1[18] := HwInputs.Reader_Operation_Result_Status_1[18];
	PlcInputs.Reader_Operation_Result_Status_1[19] := HwInputs.Reader_Operation_Result_Status_1[19];
	PlcInputs.Reader_Read_Data_128Byte_1[0] := HwInputs.Reader_Read_Data_128Byte_1[0];
	PlcInputs.Reader_Read_Data_128Byte_1[1] := HwInputs.Reader_Read_Data_128Byte_1[1];
	PlcInputs.Reader_Read_Data_128Byte_1[2] := HwInputs.Reader_Read_Data_128Byte_1[2];
	PlcInputs.Reader_Read_Data_128Byte_1[3] := HwInputs.Reader_Read_Data_128Byte_1[3];
	PlcInputs.Reader_Read_Data_128Byte_1[4] := HwInputs.Reader_Read_Data_128Byte_1[4];
	PlcInputs.Reader_Read_Data_128Byte_1[5] := HwInputs.Reader_Read_Data_128Byte_1[5];
	PlcInputs.Reader_Read_Data_128Byte_1[6] := HwInputs.Reader_Read_Data_128Byte_1[6];
	PlcInputs.Reader_Read_Data_128Byte_1[7] := HwInputs.Reader_Read_Data_128Byte_1[7];
	PlcInputs.Reader_Read_Data_128Byte_1[8] := HwInputs.Reader_Read_Data_128Byte_1[8];
	PlcInputs.Reader_Read_Data_128Byte_1[9] := HwInputs.Reader_Read_Data_128Byte_1[9];
	PlcInputs.Reader_Read_Data_128Byte_1[10] := HwInputs.Reader_Read_Data_128Byte_1[10];
	PlcInputs.Reader_Read_Data_128Byte_1[11] := HwInputs.Reader_Read_Data_128Byte_1[11];
	PlcInputs.Reader_Read_Data_128Byte_1[12] := HwInputs.Reader_Read_Data_128Byte_1[12];
	PlcInputs.Reader_Read_Data_128Byte_1[13] := HwInputs.Reader_Read_Data_128Byte_1[13];
	PlcInputs.Reader_Read_Data_128Byte_1[14] := HwInputs.Reader_Read_Data_128Byte_1[14];
	PlcInputs.Reader_Read_Data_128Byte_1[15] := HwInputs.Reader_Read_Data_128Byte_1[15];
	PlcInputs.Reader_Read_Data_128Byte_1[16] := HwInputs.Reader_Read_Data_128Byte_1[16];
	PlcInputs.Reader_Read_Data_128Byte_1[17] := HwInputs.Reader_Read_Data_128Byte_1[17];
	PlcInputs.Reader_Read_Data_128Byte_1[18] := HwInputs.Reader_Read_Data_128Byte_1[18];
	PlcInputs.Reader_Read_Data_128Byte_1[19] := HwInputs.Reader_Read_Data_128Byte_1[19];
	PlcInputs.Reader_Read_Data_128Byte_1[20] := HwInputs.Reader_Read_Data_128Byte_1[20];
	PlcInputs.Reader_Read_Data_128Byte_1[21] := HwInputs.Reader_Read_Data_128Byte_1[21];
	PlcInputs.Reader_Read_Data_128Byte_1[22] := HwInputs.Reader_Read_Data_128Byte_1[22];
	PlcInputs.Reader_Read_Data_128Byte_1[23] := HwInputs.Reader_Read_Data_128Byte_1[23];
	PlcInputs.Reader_Read_Data_128Byte_1[24] := HwInputs.Reader_Read_Data_128Byte_1[24];
	PlcInputs.Reader_Read_Data_128Byte_1[25] := HwInputs.Reader_Read_Data_128Byte_1[25];
	PlcInputs.Reader_Read_Data_128Byte_1[26] := HwInputs.Reader_Read_Data_128Byte_1[26];
	PlcInputs.Reader_Read_Data_128Byte_1[27] := HwInputs.Reader_Read_Data_128Byte_1[27];
	PlcInputs.Reader_Read_Data_128Byte_1[28] := HwInputs.Reader_Read_Data_128Byte_1[28];
	PlcInputs.Reader_Read_Data_128Byte_1[29] := HwInputs.Reader_Read_Data_128Byte_1[29];
	PlcInputs.Reader_Read_Data_128Byte_1[30] := HwInputs.Reader_Read_Data_128Byte_1[30];
	PlcInputs.Reader_Read_Data_128Byte_1[31] := HwInputs.Reader_Read_Data_128Byte_1[31];
	PlcInputs.Reader_Read_Data_128Byte_1[32] := HwInputs.Reader_Read_Data_128Byte_1[32];
	PlcInputs.Reader_Read_Data_128Byte_1[33] := HwInputs.Reader_Read_Data_128Byte_1[33];
	PlcInputs.Reader_Read_Data_128Byte_1[34] := HwInputs.Reader_Read_Data_128Byte_1[34];
	PlcInputs.Reader_Read_Data_128Byte_1[35] := HwInputs.Reader_Read_Data_128Byte_1[35];
	PlcInputs.Reader_Read_Data_128Byte_1[36] := HwInputs.Reader_Read_Data_128Byte_1[36];
	PlcInputs.Reader_Read_Data_128Byte_1[37] := HwInputs.Reader_Read_Data_128Byte_1[37];
	PlcInputs.Reader_Read_Data_128Byte_1[38] := HwInputs.Reader_Read_Data_128Byte_1[38];
	PlcInputs.Reader_Read_Data_128Byte_1[39] := HwInputs.Reader_Read_Data_128Byte_1[39];
	PlcInputs.Reader_Read_Data_128Byte_1[40] := HwInputs.Reader_Read_Data_128Byte_1[40];
	PlcInputs.Reader_Read_Data_128Byte_1[41] := HwInputs.Reader_Read_Data_128Byte_1[41];
	PlcInputs.Reader_Read_Data_128Byte_1[42] := HwInputs.Reader_Read_Data_128Byte_1[42];
	PlcInputs.Reader_Read_Data_128Byte_1[43] := HwInputs.Reader_Read_Data_128Byte_1[43];
	PlcInputs.Reader_Read_Data_128Byte_1[44] := HwInputs.Reader_Read_Data_128Byte_1[44];
	PlcInputs.Reader_Read_Data_128Byte_1[45] := HwInputs.Reader_Read_Data_128Byte_1[45];
	PlcInputs.Reader_Read_Data_128Byte_1[46] := HwInputs.Reader_Read_Data_128Byte_1[46];
	PlcInputs.Reader_Read_Data_128Byte_1[47] := HwInputs.Reader_Read_Data_128Byte_1[47];
	PlcInputs.Reader_Read_Data_128Byte_1[48] := HwInputs.Reader_Read_Data_128Byte_1[48];
	PlcInputs.Reader_Read_Data_128Byte_1[49] := HwInputs.Reader_Read_Data_128Byte_1[49];
	PlcInputs.Reader_Read_Data_128Byte_1[50] := HwInputs.Reader_Read_Data_128Byte_1[50];
	PlcInputs.Reader_Read_Data_128Byte_1[51] := HwInputs.Reader_Read_Data_128Byte_1[51];
	PlcInputs.Reader_Read_Data_128Byte_1[52] := HwInputs.Reader_Read_Data_128Byte_1[52];
	PlcInputs.Reader_Read_Data_128Byte_1[53] := HwInputs.Reader_Read_Data_128Byte_1[53];
	PlcInputs.Reader_Read_Data_128Byte_1[54] := HwInputs.Reader_Read_Data_128Byte_1[54];
	PlcInputs.Reader_Read_Data_128Byte_1[55] := HwInputs.Reader_Read_Data_128Byte_1[55];
	PlcInputs.Reader_Read_Data_128Byte_1[56] := HwInputs.Reader_Read_Data_128Byte_1[56];
	PlcInputs.Reader_Read_Data_128Byte_1[57] := HwInputs.Reader_Read_Data_128Byte_1[57];
	PlcInputs.Reader_Read_Data_128Byte_1[58] := HwInputs.Reader_Read_Data_128Byte_1[58];
	PlcInputs.Reader_Read_Data_128Byte_1[59] := HwInputs.Reader_Read_Data_128Byte_1[59];
	PlcInputs.Reader_Read_Data_128Byte_1[60] := HwInputs.Reader_Read_Data_128Byte_1[60];
	PlcInputs.Reader_Read_Data_128Byte_1[61] := HwInputs.Reader_Read_Data_128Byte_1[61];
	PlcInputs.Reader_Read_Data_128Byte_1[62] := HwInputs.Reader_Read_Data_128Byte_1[62];
	PlcInputs.Reader_Read_Data_128Byte_1[63] := HwInputs.Reader_Read_Data_128Byte_1[63];
	PlcInputs.Reader_Read_Data_128Byte_1[64] := HwInputs.Reader_Read_Data_128Byte_1[64];
	PlcInputs.Reader_Read_Data_128Byte_1[65] := HwInputs.Reader_Read_Data_128Byte_1[65];
	PlcInputs.Reader_Read_Data_128Byte_1[66] := HwInputs.Reader_Read_Data_128Byte_1[66];
	PlcInputs.Reader_Read_Data_128Byte_1[67] := HwInputs.Reader_Read_Data_128Byte_1[67];
	PlcInputs.Reader_Read_Data_128Byte_1[68] := HwInputs.Reader_Read_Data_128Byte_1[68];
	PlcInputs.Reader_Read_Data_128Byte_1[69] := HwInputs.Reader_Read_Data_128Byte_1[69];
	PlcInputs.Reader_Read_Data_128Byte_1[70] := HwInputs.Reader_Read_Data_128Byte_1[70];
	PlcInputs.Reader_Read_Data_128Byte_1[71] := HwInputs.Reader_Read_Data_128Byte_1[71];
	PlcInputs.Reader_Read_Data_128Byte_1[72] := HwInputs.Reader_Read_Data_128Byte_1[72];
	PlcInputs.Reader_Read_Data_128Byte_1[73] := HwInputs.Reader_Read_Data_128Byte_1[73];
	PlcInputs.Reader_Read_Data_128Byte_1[74] := HwInputs.Reader_Read_Data_128Byte_1[74];
	PlcInputs.Reader_Read_Data_128Byte_1[75] := HwInputs.Reader_Read_Data_128Byte_1[75];
	PlcInputs.Reader_Read_Data_128Byte_1[76] := HwInputs.Reader_Read_Data_128Byte_1[76];
	PlcInputs.Reader_Read_Data_128Byte_1[77] := HwInputs.Reader_Read_Data_128Byte_1[77];
	PlcInputs.Reader_Read_Data_128Byte_1[78] := HwInputs.Reader_Read_Data_128Byte_1[78];
	PlcInputs.Reader_Read_Data_128Byte_1[79] := HwInputs.Reader_Read_Data_128Byte_1[79];
	PlcInputs.Reader_Read_Data_128Byte_1[80] := HwInputs.Reader_Read_Data_128Byte_1[80];
	PlcInputs.Reader_Read_Data_128Byte_1[81] := HwInputs.Reader_Read_Data_128Byte_1[81];
	PlcInputs.Reader_Read_Data_128Byte_1[82] := HwInputs.Reader_Read_Data_128Byte_1[82];
	PlcInputs.Reader_Read_Data_128Byte_1[83] := HwInputs.Reader_Read_Data_128Byte_1[83];
	PlcInputs.Reader_Read_Data_128Byte_1[84] := HwInputs.Reader_Read_Data_128Byte_1[84];
	PlcInputs.Reader_Read_Data_128Byte_1[85] := HwInputs.Reader_Read_Data_128Byte_1[85];
	PlcInputs.Reader_Read_Data_128Byte_1[86] := HwInputs.Reader_Read_Data_128Byte_1[86];
	PlcInputs.Reader_Read_Data_128Byte_1[87] := HwInputs.Reader_Read_Data_128Byte_1[87];
	PlcInputs.Reader_Read_Data_128Byte_1[88] := HwInputs.Reader_Read_Data_128Byte_1[88];
	PlcInputs.Reader_Read_Data_128Byte_1[89] := HwInputs.Reader_Read_Data_128Byte_1[89];
	PlcInputs.Reader_Read_Data_128Byte_1[90] := HwInputs.Reader_Read_Data_128Byte_1[90];
	PlcInputs.Reader_Read_Data_128Byte_1[91] := HwInputs.Reader_Read_Data_128Byte_1[91];
	PlcInputs.Reader_Read_Data_128Byte_1[92] := HwInputs.Reader_Read_Data_128Byte_1[92];
	PlcInputs.Reader_Read_Data_128Byte_1[93] := HwInputs.Reader_Read_Data_128Byte_1[93];
	PlcInputs.Reader_Read_Data_128Byte_1[94] := HwInputs.Reader_Read_Data_128Byte_1[94];
	PlcInputs.Reader_Read_Data_128Byte_1[95] := HwInputs.Reader_Read_Data_128Byte_1[95];
	PlcInputs.Reader_Read_Data_128Byte_1[96] := HwInputs.Reader_Read_Data_128Byte_1[96];
	PlcInputs.Reader_Read_Data_128Byte_1[97] := HwInputs.Reader_Read_Data_128Byte_1[97];
	PlcInputs.Reader_Read_Data_128Byte_1[98] := HwInputs.Reader_Read_Data_128Byte_1[98];
	PlcInputs.Reader_Read_Data_128Byte_1[99] := HwInputs.Reader_Read_Data_128Byte_1[99];
	PlcInputs.Reader_Read_Data_128Byte_1[100] := HwInputs.Reader_Read_Data_128Byte_1[100];
	PlcInputs.Reader_Read_Data_128Byte_1[101] := HwInputs.Reader_Read_Data_128Byte_1[101];
	PlcInputs.Reader_Read_Data_128Byte_1[102] := HwInputs.Reader_Read_Data_128Byte_1[102];
	PlcInputs.Reader_Read_Data_128Byte_1[103] := HwInputs.Reader_Read_Data_128Byte_1[103];
	PlcInputs.Reader_Read_Data_128Byte_1[104] := HwInputs.Reader_Read_Data_128Byte_1[104];
	PlcInputs.Reader_Read_Data_128Byte_1[105] := HwInputs.Reader_Read_Data_128Byte_1[105];
	PlcInputs.Reader_Read_Data_128Byte_1[106] := HwInputs.Reader_Read_Data_128Byte_1[106];
	PlcInputs.Reader_Read_Data_128Byte_1[107] := HwInputs.Reader_Read_Data_128Byte_1[107];
	PlcInputs.Reader_Read_Data_128Byte_1[108] := HwInputs.Reader_Read_Data_128Byte_1[108];
	PlcInputs.Reader_Read_Data_128Byte_1[109] := HwInputs.Reader_Read_Data_128Byte_1[109];
	PlcInputs.Reader_Read_Data_128Byte_1[110] := HwInputs.Reader_Read_Data_128Byte_1[110];
	PlcInputs.Reader_Read_Data_128Byte_1[111] := HwInputs.Reader_Read_Data_128Byte_1[111];
	PlcInputs.Reader_Read_Data_128Byte_1[112] := HwInputs.Reader_Read_Data_128Byte_1[112];
	PlcInputs.Reader_Read_Data_128Byte_1[113] := HwInputs.Reader_Read_Data_128Byte_1[113];
	PlcInputs.Reader_Read_Data_128Byte_1[114] := HwInputs.Reader_Read_Data_128Byte_1[114];
	PlcInputs.Reader_Read_Data_128Byte_1[115] := HwInputs.Reader_Read_Data_128Byte_1[115];
	PlcInputs.Reader_Read_Data_128Byte_1[116] := HwInputs.Reader_Read_Data_128Byte_1[116];
	PlcInputs.Reader_Read_Data_128Byte_1[117] := HwInputs.Reader_Read_Data_128Byte_1[117];
	PlcInputs.Reader_Read_Data_128Byte_1[118] := HwInputs.Reader_Read_Data_128Byte_1[118];
	PlcInputs.Reader_Read_Data_128Byte_1[119] := HwInputs.Reader_Read_Data_128Byte_1[119];
	PlcInputs.Reader_Read_Data_128Byte_1[120] := HwInputs.Reader_Read_Data_128Byte_1[120];
	PlcInputs.Reader_Read_Data_128Byte_1[121] := HwInputs.Reader_Read_Data_128Byte_1[121];
	PlcInputs.Reader_Read_Data_128Byte_1[122] := HwInputs.Reader_Read_Data_128Byte_1[122];
	PlcInputs.Reader_Read_Data_128Byte_1[123] := HwInputs.Reader_Read_Data_128Byte_1[123];
	PlcInputs.Reader_Read_Data_128Byte_1[124] := HwInputs.Reader_Read_Data_128Byte_1[124];
	PlcInputs.Reader_Read_Data_128Byte_1[125] := HwInputs.Reader_Read_Data_128Byte_1[125];
	PlcInputs.Reader_Read_Data_128Byte_1[126] := HwInputs.Reader_Read_Data_128Byte_1[126];
	PlcInputs.Reader_Read_Data_128Byte_1[127] := HwInputs.Reader_Read_Data_128Byte_1[127];
	PlcInputs.Reader_Read_Data_128Byte_1[128] := HwInputs.Reader_Read_Data_128Byte_1[128];
	PlcInputs.Reader_Read_Data_128Byte_1[129] := HwInputs.Reader_Read_Data_128Byte_1[129];
	PlcInputs.Reader_Read_Data_128Byte_1[130] := HwInputs.Reader_Read_Data_128Byte_1[130];
	PlcInputs.Reader_Read_Data_128Byte_1[131] := HwInputs.Reader_Read_Data_128Byte_1[131];
	PlcInputs.Reader_Read_Data_128Byte_1[132] := HwInputs.Reader_Read_Data_128Byte_1[132];
	PlcInputs.Reader_Read_Data_128Byte_1[133] := HwInputs.Reader_Read_Data_128Byte_1[133];
	PlcInputs.Reader_Read_Data_128Byte_1[134] := HwInputs.Reader_Read_Data_128Byte_1[134];
	PlcInputs.Reader_Read_Data_128Byte_1[135] := HwInputs.Reader_Read_Data_128Byte_1[135];
END_FUNCTION

(* ---- CopyOutputs.st ---- *)
FUNCTION CopyOutputs
	VAR_EXTERNAL
		HwOutputs : HwOutputs;
		PlcOutputs : PlcOutputs;
	END_VAR
	HwOutputs.A6_15A5 := PlcOutputs.A6_15A5;
	HwOutputs.A6_15A6 := PlcOutputs.A6_15A6;
	HwOutputs.A6_15A7 := PlcOutputs.A6_15A7;
	HwOutputs.A6_15A8 := PlcOutputs.A6_15A8;
	HwOutputs.A6_15A10[0] := PlcOutputs.A6_15A10[0];
	HwOutputs.A6_15A10[1] := PlcOutputs.A6_15A10[1];
	HwOutputs.A6_15A10[2] := PlcOutputs.A6_15A10[2];
	HwOutputs.A6_15A10[3] := PlcOutputs.A6_15A10[3];
	HwOutputs.A6_15A10[4] := PlcOutputs.A6_15A10[4];
	HwOutputs.A6_15A10[5] := PlcOutputs.A6_15A10[5];
	HwOutputs.A6_15A10[6] := PlcOutputs.A6_15A10[6];
	HwOutputs.A6_15A10[7] := PlcOutputs.A6_15A10[7];
	HwOutputs.VI_13_MPA1S_VMPA1_FB_EMS_8_8DO_1 := PlcOutputs.VI_13_MPA1S_VMPA1_FB_EMS_8_8DO_1;
	HwOutputs.VI_13_MPA1S_VMPA1_FB_EMS_8_8DO_2 := PlcOutputs.VI_13_MPA1S_VMPA1_FB_EMS_8_8DO_2;
	HwOutputs.VI_13_MPA1S_VMPA1_FB_EMS_8_8DO_3 := PlcOutputs.VI_13_MPA1S_VMPA1_FB_EMS_8_8DO_3;
	HwOutputs.VI_13_MPA1S_VMPA1_FB_EMS_8_8DO_4 := PlcOutputs.VI_13_MPA1S_VMPA1_FB_EMS_8_8DO_4;
	HwOutputs.VI_13_MPA1S_VMPA1_FB_EMS_8_8DO_5 := PlcOutputs.VI_13_MPA1S_VMPA1_FB_EMS_8_8DO_5;
	HwOutputs.VI_13_MPA1S_VMPA1_FB_EMS_8_8DO_6 := PlcOutputs.VI_13_MPA1S_VMPA1_FB_EMS_8_8DO_6;
	HwOutputs.VI_13_MPA1S_VMPA1_FB_EMS_8_8DO_7 := PlcOutputs.VI_13_MPA1S_VMPA1_FB_EMS_8_8DO_7;
	HwOutputs.VI_13_MPA1S_VMPA1_FB_EMS_8_8DO_8 := PlcOutputs.VI_13_MPA1S_VMPA1_FB_EMS_8_8DO_8;
	HwOutputs.Bash_Output_1_byte_1 := PlcOutputs.Bash_Output_1_byte_1;
	HwOutputs.Bash_Output_1_byte_2 := PlcOutputs.Bash_Output_1_byte_2;
	HwOutputs.AEBDown_Output_1_byte_1 := PlcOutputs.AEBDown_Output_1_byte_1;
	HwOutputs.AEBDown_Output_1_byte_2 := PlcOutputs.AEBDown_Output_1_byte_2;
	HwOutputs.AEBUp_Output_1_byte_1 := PlcOutputs.AEBUp_Output_1_byte_1;
	HwOutputs.AEBUp_Output_1_byte_2 := PlcOutputs.AEBUp_Output_1_byte_2;
	HwOutputs.AETDown_Output_1_byte_1 := PlcOutputs.AETDown_Output_1_byte_1;
	HwOutputs.AETDown_Output_1_byte_2 := PlcOutputs.AETDown_Output_1_byte_2;
	HwOutputs.AETUp_Output_1_byte_1 := PlcOutputs.AETUp_Output_1_byte_1;
	HwOutputs.AETUp_Output_1_byte_2 := PlcOutputs.AETUp_Output_1_byte_2;
	HwOutputs.GT2_DL_PN1_1 := PlcOutputs.GT2_DL_PN1_1;
	HwOutputs.GT2_B1 := PlcOutputs.GT2_B1;
	HwOutputs.GT2_B2 := PlcOutputs.GT2_B2;
	HwOutputs.GT2_B3 := PlcOutputs.GT2_B3;
	HwOutputs.GT2_B4 := PlcOutputs.GT2_B4;
	HwOutputs.GT2_B5 := PlcOutputs.GT2_B5;
	HwOutputs.GT2_B6 := PlcOutputs.GT2_B6;
	HwOutputs.GT2_B7 := PlcOutputs.GT2_B7;
	HwOutputs.GT2_B8 := PlcOutputs.GT2_B8;
	HwOutputs.GT2_B9 := PlcOutputs.GT2_B9;
	HwOutputs.CPX_CW_SW := PlcOutputs.CPX_CW_SW;
	HwOutputs.CPX_CNC[0] := PlcOutputs.CPX_CNC[0];
	HwOutputs.CPX_CNC[1] := PlcOutputs.CPX_CNC[1];
	HwOutputs.CPX_CNC[2] := PlcOutputs.CPX_CNC[2];
	HwOutputs.CPX_CNC[3] := PlcOutputs.CPX_CNC[3];
	HwOutputs.CPX_CNC[4] := PlcOutputs.CPX_CNC[4];
	HwOutputs.CPX_CNC[5] := PlcOutputs.CPX_CNC[5];
	HwOutputs.CPX_CNC[6] := PlcOutputs.CPX_CNC[6];
	HwOutputs.CPX_CNC[7] := PlcOutputs.CPX_CNC[7];
	HwOutputs.CPX_CNC[8] := PlcOutputs.CPX_CNC[8];
	HwOutputs.CPX_CNC[9] := PlcOutputs.CPX_CNC[9];
	HwOutputs.CPX_CNC[10] := PlcOutputs.CPX_CNC[10];
	HwOutputs.CPX_CNC[11] := PlcOutputs.CPX_CNC[11];
	HwOutputs.CPX_CNC[12] := PlcOutputs.CPX_CNC[12];
	HwOutputs.CPX_CNC[13] := PlcOutputs.CPX_CNC[13];
	HwOutputs.CPX_CNC[14] := PlcOutputs.CPX_CNC[14];
	HwOutputs.CPX_CNC[15] := PlcOutputs.CPX_CNC[15];
	HwOutputs.CPX_CNC[16] := PlcOutputs.CPX_CNC[16];
	HwOutputs.CPX_CNC[17] := PlcOutputs.CPX_CNC[17];
	HwOutputs.CPX_CNC[18] := PlcOutputs.CPX_CNC[18];
	HwOutputs.CPX_CNC[19] := PlcOutputs.CPX_CNC[19];
	HwOutputs.CPX_CNC[20] := PlcOutputs.CPX_CNC[20];
	HwOutputs.CPX_CNC[21] := PlcOutputs.CPX_CNC[21];
	HwOutputs.CPX_CNC[22] := PlcOutputs.CPX_CNC[22];
	HwOutputs.CPX_CNC[23] := PlcOutputs.CPX_CNC[23];
	HwOutputs.CPX_CNC[24] := PlcOutputs.CPX_CNC[24];
	HwOutputs.CPX_CNC[25] := PlcOutputs.CPX_CNC[25];
	HwOutputs.CPX_CNC[26] := PlcOutputs.CPX_CNC[26];
	HwOutputs.CPX_CNC[27] := PlcOutputs.CPX_CNC[27];
	HwOutputs.CPX_CNC[28] := PlcOutputs.CPX_CNC[28];
	HwOutputs.CPX_CNC[29] := PlcOutputs.CPX_CNC[29];
	HwOutputs.CPX_CNC[30] := PlcOutputs.CPX_CNC[30];
	HwOutputs.CPX_CNC[31] := PlcOutputs.CPX_CNC[31];
	HwOutputs.CPX_PtP[0] := PlcOutputs.CPX_PtP[0];
	HwOutputs.CPX_PtP[1] := PlcOutputs.CPX_PtP[1];
	HwOutputs.CPX_PtP[2] := PlcOutputs.CPX_PtP[2];
	HwOutputs.CPX_PtP[3] := PlcOutputs.CPX_PtP[3];
	HwOutputs.CPX_PtP[4] := PlcOutputs.CPX_PtP[4];
	HwOutputs.CPX_PtP[5] := PlcOutputs.CPX_PtP[5];
	HwOutputs.CPX_PtP[6] := PlcOutputs.CPX_PtP[6];
	HwOutputs.CPX_PtP[7] := PlcOutputs.CPX_PtP[7];
	HwOutputs.CPX_PtP[8] := PlcOutputs.CPX_PtP[8];
	HwOutputs.CPX_PtP[9] := PlcOutputs.CPX_PtP[9];
	HwOutputs.CPX_PtP[10] := PlcOutputs.CPX_PtP[10];
	HwOutputs.CPX_PtP[11] := PlcOutputs.CPX_PtP[11];
	HwOutputs.CPX_PtP[12] := PlcOutputs.CPX_PtP[12];
	HwOutputs.CPX_PtP[13] := PlcOutputs.CPX_PtP[13];
	HwOutputs.CPX_PtP[14] := PlcOutputs.CPX_PtP[14];
	HwOutputs.CPX_PtP[15] := PlcOutputs.CPX_PtP[15];
	HwOutputs.CPX_Error[0] := PlcOutputs.CPX_Error[0];
	HwOutputs.CPX_Error[1] := PlcOutputs.CPX_Error[1];
	HwOutputs.CPX_Error[2] := PlcOutputs.CPX_Error[2];
	HwOutputs.CPX_Error[3] := PlcOutputs.CPX_Error[3];
	HwOutputs.CPX_Error[4] := PlcOutputs.CPX_Error[4];
	HwOutputs.CPX_Error[5] := PlcOutputs.CPX_Error[5];
	HwOutputs.CPX_Error[6] := PlcOutputs.CPX_Error[6];
	HwOutputs.CPX_Error[7] := PlcOutputs.CPX_Error[7];
	HwOutputs.CPX_Error[8] := PlcOutputs.CPX_Error[8];
	HwOutputs.CPX_Error[9] := PlcOutputs.CPX_Error[9];
	HwOutputs.CPX_Error[10] := PlcOutputs.CPX_Error[10];
	HwOutputs.CPX_Error[11] := PlcOutputs.CPX_Error[11];
	HwOutputs.CPX_Error[12] := PlcOutputs.CPX_Error[12];
	HwOutputs.CPX_Error[13] := PlcOutputs.CPX_Error[13];
	HwOutputs.CPX_Error[14] := PlcOutputs.CPX_Error[14];
	HwOutputs.CPX_Error[15] := PlcOutputs.CPX_Error[15];
	HwOutputs.CPX_Error[16] := PlcOutputs.CPX_Error[16];
	HwOutputs.CPX_Error[17] := PlcOutputs.CPX_Error[17];
	HwOutputs.CPX_Error[18] := PlcOutputs.CPX_Error[18];
	HwOutputs.CPX_Error[19] := PlcOutputs.CPX_Error[19];
	HwOutputs.CPX_Error[20] := PlcOutputs.CPX_Error[20];
	HwOutputs.CPX_Error[21] := PlcOutputs.CPX_Error[21];
	HwOutputs.CPX_Error[22] := PlcOutputs.CPX_Error[22];
	HwOutputs.CPX_Error[23] := PlcOutputs.CPX_Error[23];
	HwOutputs.CPX_Error[24] := PlcOutputs.CPX_Error[24];
	HwOutputs.CPX_Error[25] := PlcOutputs.CPX_Error[25];
	HwOutputs.CPX_Error[26] := PlcOutputs.CPX_Error[26];
	HwOutputs.CPX_Error[27] := PlcOutputs.CPX_Error[27];
	HwOutputs.CPX_Error[28] := PlcOutputs.CPX_Error[28];
	HwOutputs.CPX_Error[29] := PlcOutputs.CPX_Error[29];
	HwOutputs.CPX_Error[30] := PlcOutputs.CPX_Error[30];
	HwOutputs.CPX_Error[31] := PlcOutputs.CPX_Error[31];
	HwOutputs.Reader_Latch_and_Error_Clear_Control_Bits_1 := PlcOutputs.Reader_Latch_and_Error_Clear_Control_Bits_1;
	HwOutputs.Reader_Operation_instruction_Control_Bits_1 := PlcOutputs.Reader_Operation_instruction_Control_Bits_1;
	HwOutputs.Reader_Completion_Clear_Control_Bits_1 := PlcOutputs.Reader_Completion_Clear_Control_Bits_1;
	HwOutputs.Reader_Parameter_Bank_Number_1 := PlcOutputs.Reader_Parameter_Bank_Number_1;
	HwOutputs.Reader_User_Data_128Byte_1[0] := PlcOutputs.Reader_User_Data_128Byte_1[0];
	HwOutputs.Reader_User_Data_128Byte_1[1] := PlcOutputs.Reader_User_Data_128Byte_1[1];
	HwOutputs.Reader_User_Data_128Byte_1[2] := PlcOutputs.Reader_User_Data_128Byte_1[2];
	HwOutputs.Reader_User_Data_128Byte_1[3] := PlcOutputs.Reader_User_Data_128Byte_1[3];
	HwOutputs.Reader_User_Data_128Byte_1[4] := PlcOutputs.Reader_User_Data_128Byte_1[4];
	HwOutputs.Reader_User_Data_128Byte_1[5] := PlcOutputs.Reader_User_Data_128Byte_1[5];
	HwOutputs.Reader_User_Data_128Byte_1[6] := PlcOutputs.Reader_User_Data_128Byte_1[6];
	HwOutputs.Reader_User_Data_128Byte_1[7] := PlcOutputs.Reader_User_Data_128Byte_1[7];
	HwOutputs.Reader_User_Data_128Byte_1[8] := PlcOutputs.Reader_User_Data_128Byte_1[8];
	HwOutputs.Reader_User_Data_128Byte_1[9] := PlcOutputs.Reader_User_Data_128Byte_1[9];
	HwOutputs.Reader_User_Data_128Byte_1[10] := PlcOutputs.Reader_User_Data_128Byte_1[10];
	HwOutputs.Reader_User_Data_128Byte_1[11] := PlcOutputs.Reader_User_Data_128Byte_1[11];
	HwOutputs.Reader_User_Data_128Byte_1[12] := PlcOutputs.Reader_User_Data_128Byte_1[12];
	HwOutputs.Reader_User_Data_128Byte_1[13] := PlcOutputs.Reader_User_Data_128Byte_1[13];
	HwOutputs.Reader_User_Data_128Byte_1[14] := PlcOutputs.Reader_User_Data_128Byte_1[14];
	HwOutputs.Reader_User_Data_128Byte_1[15] := PlcOutputs.Reader_User_Data_128Byte_1[15];
	HwOutputs.Reader_User_Data_128Byte_1[16] := PlcOutputs.Reader_User_Data_128Byte_1[16];
	HwOutputs.Reader_User_Data_128Byte_1[17] := PlcOutputs.Reader_User_Data_128Byte_1[17];
	HwOutputs.Reader_User_Data_128Byte_1[18] := PlcOutputs.Reader_User_Data_128Byte_1[18];
	HwOutputs.Reader_User_Data_128Byte_1[19] := PlcOutputs.Reader_User_Data_128Byte_1[19];
	HwOutputs.Reader_User_Data_128Byte_1[20] := PlcOutputs.Reader_User_Data_128Byte_1[20];
	HwOutputs.Reader_User_Data_128Byte_1[21] := PlcOutputs.Reader_User_Data_128Byte_1[21];
	HwOutputs.Reader_User_Data_128Byte_1[22] := PlcOutputs.Reader_User_Data_128Byte_1[22];
	HwOutputs.Reader_User_Data_128Byte_1[23] := PlcOutputs.Reader_User_Data_128Byte_1[23];
	HwOutputs.Reader_User_Data_128Byte_1[24] := PlcOutputs.Reader_User_Data_128Byte_1[24];
	HwOutputs.Reader_User_Data_128Byte_1[25] := PlcOutputs.Reader_User_Data_128Byte_1[25];
	HwOutputs.Reader_User_Data_128Byte_1[26] := PlcOutputs.Reader_User_Data_128Byte_1[26];
	HwOutputs.Reader_User_Data_128Byte_1[27] := PlcOutputs.Reader_User_Data_128Byte_1[27];
	HwOutputs.Reader_User_Data_128Byte_1[28] := PlcOutputs.Reader_User_Data_128Byte_1[28];
	HwOutputs.Reader_User_Data_128Byte_1[29] := PlcOutputs.Reader_User_Data_128Byte_1[29];
	HwOutputs.Reader_User_Data_128Byte_1[30] := PlcOutputs.Reader_User_Data_128Byte_1[30];
	HwOutputs.Reader_User_Data_128Byte_1[31] := PlcOutputs.Reader_User_Data_128Byte_1[31];
	HwOutputs.Reader_User_Data_128Byte_1[32] := PlcOutputs.Reader_User_Data_128Byte_1[32];
	HwOutputs.Reader_User_Data_128Byte_1[33] := PlcOutputs.Reader_User_Data_128Byte_1[33];
	HwOutputs.Reader_User_Data_128Byte_1[34] := PlcOutputs.Reader_User_Data_128Byte_1[34];
	HwOutputs.Reader_User_Data_128Byte_1[35] := PlcOutputs.Reader_User_Data_128Byte_1[35];
	HwOutputs.Reader_User_Data_128Byte_1[36] := PlcOutputs.Reader_User_Data_128Byte_1[36];
	HwOutputs.Reader_User_Data_128Byte_1[37] := PlcOutputs.Reader_User_Data_128Byte_1[37];
	HwOutputs.Reader_User_Data_128Byte_1[38] := PlcOutputs.Reader_User_Data_128Byte_1[38];
	HwOutputs.Reader_User_Data_128Byte_1[39] := PlcOutputs.Reader_User_Data_128Byte_1[39];
	HwOutputs.Reader_User_Data_128Byte_1[40] := PlcOutputs.Reader_User_Data_128Byte_1[40];
	HwOutputs.Reader_User_Data_128Byte_1[41] := PlcOutputs.Reader_User_Data_128Byte_1[41];
	HwOutputs.Reader_User_Data_128Byte_1[42] := PlcOutputs.Reader_User_Data_128Byte_1[42];
	HwOutputs.Reader_User_Data_128Byte_1[43] := PlcOutputs.Reader_User_Data_128Byte_1[43];
	HwOutputs.Reader_User_Data_128Byte_1[44] := PlcOutputs.Reader_User_Data_128Byte_1[44];
	HwOutputs.Reader_User_Data_128Byte_1[45] := PlcOutputs.Reader_User_Data_128Byte_1[45];
	HwOutputs.Reader_User_Data_128Byte_1[46] := PlcOutputs.Reader_User_Data_128Byte_1[46];
	HwOutputs.Reader_User_Data_128Byte_1[47] := PlcOutputs.Reader_User_Data_128Byte_1[47];
	HwOutputs.Reader_User_Data_128Byte_1[48] := PlcOutputs.Reader_User_Data_128Byte_1[48];
	HwOutputs.Reader_User_Data_128Byte_1[49] := PlcOutputs.Reader_User_Data_128Byte_1[49];
	HwOutputs.Reader_User_Data_128Byte_1[50] := PlcOutputs.Reader_User_Data_128Byte_1[50];
	HwOutputs.Reader_User_Data_128Byte_1[51] := PlcOutputs.Reader_User_Data_128Byte_1[51];
	HwOutputs.Reader_User_Data_128Byte_1[52] := PlcOutputs.Reader_User_Data_128Byte_1[52];
	HwOutputs.Reader_User_Data_128Byte_1[53] := PlcOutputs.Reader_User_Data_128Byte_1[53];
	HwOutputs.Reader_User_Data_128Byte_1[54] := PlcOutputs.Reader_User_Data_128Byte_1[54];
	HwOutputs.Reader_User_Data_128Byte_1[55] := PlcOutputs.Reader_User_Data_128Byte_1[55];
	HwOutputs.Reader_User_Data_128Byte_1[56] := PlcOutputs.Reader_User_Data_128Byte_1[56];
	HwOutputs.Reader_User_Data_128Byte_1[57] := PlcOutputs.Reader_User_Data_128Byte_1[57];
	HwOutputs.Reader_User_Data_128Byte_1[58] := PlcOutputs.Reader_User_Data_128Byte_1[58];
	HwOutputs.Reader_User_Data_128Byte_1[59] := PlcOutputs.Reader_User_Data_128Byte_1[59];
	HwOutputs.Reader_User_Data_128Byte_1[60] := PlcOutputs.Reader_User_Data_128Byte_1[60];
	HwOutputs.Reader_User_Data_128Byte_1[61] := PlcOutputs.Reader_User_Data_128Byte_1[61];
	HwOutputs.Reader_User_Data_128Byte_1[62] := PlcOutputs.Reader_User_Data_128Byte_1[62];
	HwOutputs.Reader_User_Data_128Byte_1[63] := PlcOutputs.Reader_User_Data_128Byte_1[63];
	HwOutputs.Reader_User_Data_128Byte_1[64] := PlcOutputs.Reader_User_Data_128Byte_1[64];
	HwOutputs.Reader_User_Data_128Byte_1[65] := PlcOutputs.Reader_User_Data_128Byte_1[65];
	HwOutputs.Reader_User_Data_128Byte_1[66] := PlcOutputs.Reader_User_Data_128Byte_1[66];
	HwOutputs.Reader_User_Data_128Byte_1[67] := PlcOutputs.Reader_User_Data_128Byte_1[67];
	HwOutputs.Reader_User_Data_128Byte_1[68] := PlcOutputs.Reader_User_Data_128Byte_1[68];
	HwOutputs.Reader_User_Data_128Byte_1[69] := PlcOutputs.Reader_User_Data_128Byte_1[69];
	HwOutputs.Reader_User_Data_128Byte_1[70] := PlcOutputs.Reader_User_Data_128Byte_1[70];
	HwOutputs.Reader_User_Data_128Byte_1[71] := PlcOutputs.Reader_User_Data_128Byte_1[71];
	HwOutputs.Reader_User_Data_128Byte_1[72] := PlcOutputs.Reader_User_Data_128Byte_1[72];
	HwOutputs.Reader_User_Data_128Byte_1[73] := PlcOutputs.Reader_User_Data_128Byte_1[73];
	HwOutputs.Reader_User_Data_128Byte_1[74] := PlcOutputs.Reader_User_Data_128Byte_1[74];
	HwOutputs.Reader_User_Data_128Byte_1[75] := PlcOutputs.Reader_User_Data_128Byte_1[75];
	HwOutputs.Reader_User_Data_128Byte_1[76] := PlcOutputs.Reader_User_Data_128Byte_1[76];
	HwOutputs.Reader_User_Data_128Byte_1[77] := PlcOutputs.Reader_User_Data_128Byte_1[77];
	HwOutputs.Reader_User_Data_128Byte_1[78] := PlcOutputs.Reader_User_Data_128Byte_1[78];
	HwOutputs.Reader_User_Data_128Byte_1[79] := PlcOutputs.Reader_User_Data_128Byte_1[79];
	HwOutputs.Reader_User_Data_128Byte_1[80] := PlcOutputs.Reader_User_Data_128Byte_1[80];
	HwOutputs.Reader_User_Data_128Byte_1[81] := PlcOutputs.Reader_User_Data_128Byte_1[81];
	HwOutputs.Reader_User_Data_128Byte_1[82] := PlcOutputs.Reader_User_Data_128Byte_1[82];
	HwOutputs.Reader_User_Data_128Byte_1[83] := PlcOutputs.Reader_User_Data_128Byte_1[83];
	HwOutputs.Reader_User_Data_128Byte_1[84] := PlcOutputs.Reader_User_Data_128Byte_1[84];
	HwOutputs.Reader_User_Data_128Byte_1[85] := PlcOutputs.Reader_User_Data_128Byte_1[85];
	HwOutputs.Reader_User_Data_128Byte_1[86] := PlcOutputs.Reader_User_Data_128Byte_1[86];
	HwOutputs.Reader_User_Data_128Byte_1[87] := PlcOutputs.Reader_User_Data_128Byte_1[87];
	HwOutputs.Reader_User_Data_128Byte_1[88] := PlcOutputs.Reader_User_Data_128Byte_1[88];
	HwOutputs.Reader_User_Data_128Byte_1[89] := PlcOutputs.Reader_User_Data_128Byte_1[89];
	HwOutputs.Reader_User_Data_128Byte_1[90] := PlcOutputs.Reader_User_Data_128Byte_1[90];
	HwOutputs.Reader_User_Data_128Byte_1[91] := PlcOutputs.Reader_User_Data_128Byte_1[91];
	HwOutputs.Reader_User_Data_128Byte_1[92] := PlcOutputs.Reader_User_Data_128Byte_1[92];
	HwOutputs.Reader_User_Data_128Byte_1[93] := PlcOutputs.Reader_User_Data_128Byte_1[93];
	HwOutputs.Reader_User_Data_128Byte_1[94] := PlcOutputs.Reader_User_Data_128Byte_1[94];
	HwOutputs.Reader_User_Data_128Byte_1[95] := PlcOutputs.Reader_User_Data_128Byte_1[95];
	HwOutputs.Reader_User_Data_128Byte_1[96] := PlcOutputs.Reader_User_Data_128Byte_1[96];
	HwOutputs.Reader_User_Data_128Byte_1[97] := PlcOutputs.Reader_User_Data_128Byte_1[97];
	HwOutputs.Reader_User_Data_128Byte_1[98] := PlcOutputs.Reader_User_Data_128Byte_1[98];
	HwOutputs.Reader_User_Data_128Byte_1[99] := PlcOutputs.Reader_User_Data_128Byte_1[99];
	HwOutputs.Reader_User_Data_128Byte_1[100] := PlcOutputs.Reader_User_Data_128Byte_1[100];
	HwOutputs.Reader_User_Data_128Byte_1[101] := PlcOutputs.Reader_User_Data_128Byte_1[101];
	HwOutputs.Reader_User_Data_128Byte_1[102] := PlcOutputs.Reader_User_Data_128Byte_1[102];
	HwOutputs.Reader_User_Data_128Byte_1[103] := PlcOutputs.Reader_User_Data_128Byte_1[103];
	HwOutputs.Reader_User_Data_128Byte_1[104] := PlcOutputs.Reader_User_Data_128Byte_1[104];
	HwOutputs.Reader_User_Data_128Byte_1[105] := PlcOutputs.Reader_User_Data_128Byte_1[105];
	HwOutputs.Reader_User_Data_128Byte_1[106] := PlcOutputs.Reader_User_Data_128Byte_1[106];
	HwOutputs.Reader_User_Data_128Byte_1[107] := PlcOutputs.Reader_User_Data_128Byte_1[107];
	HwOutputs.Reader_User_Data_128Byte_1[108] := PlcOutputs.Reader_User_Data_128Byte_1[108];
	HwOutputs.Reader_User_Data_128Byte_1[109] := PlcOutputs.Reader_User_Data_128Byte_1[109];
	HwOutputs.Reader_User_Data_128Byte_1[110] := PlcOutputs.Reader_User_Data_128Byte_1[110];
	HwOutputs.Reader_User_Data_128Byte_1[111] := PlcOutputs.Reader_User_Data_128Byte_1[111];
	HwOutputs.Reader_User_Data_128Byte_1[112] := PlcOutputs.Reader_User_Data_128Byte_1[112];
	HwOutputs.Reader_User_Data_128Byte_1[113] := PlcOutputs.Reader_User_Data_128Byte_1[113];
	HwOutputs.Reader_User_Data_128Byte_1[114] := PlcOutputs.Reader_User_Data_128Byte_1[114];
	HwOutputs.Reader_User_Data_128Byte_1[115] := PlcOutputs.Reader_User_Data_128Byte_1[115];
	HwOutputs.Reader_User_Data_128Byte_1[116] := PlcOutputs.Reader_User_Data_128Byte_1[116];
	HwOutputs.Reader_User_Data_128Byte_1[117] := PlcOutputs.Reader_User_Data_128Byte_1[117];
	HwOutputs.Reader_User_Data_128Byte_1[118] := PlcOutputs.Reader_User_Data_128Byte_1[118];
	HwOutputs.Reader_User_Data_128Byte_1[119] := PlcOutputs.Reader_User_Data_128Byte_1[119];
	HwOutputs.Reader_User_Data_128Byte_1[120] := PlcOutputs.Reader_User_Data_128Byte_1[120];
	HwOutputs.Reader_User_Data_128Byte_1[121] := PlcOutputs.Reader_User_Data_128Byte_1[121];
	HwOutputs.Reader_User_Data_128Byte_1[122] := PlcOutputs.Reader_User_Data_128Byte_1[122];
	HwOutputs.Reader_User_Data_128Byte_1[123] := PlcOutputs.Reader_User_Data_128Byte_1[123];
	HwOutputs.Reader_User_Data_128Byte_1[124] := PlcOutputs.Reader_User_Data_128Byte_1[124];
	HwOutputs.Reader_User_Data_128Byte_1[125] := PlcOutputs.Reader_User_Data_128Byte_1[125];
	HwOutputs.Reader_User_Data_128Byte_1[126] := PlcOutputs.Reader_User_Data_128Byte_1[126];
	HwOutputs.Reader_User_Data_128Byte_1[127] := PlcOutputs.Reader_User_Data_128Byte_1[127];
	HwOutputs.Reader_User_Data_128Byte_1[128] := PlcOutputs.Reader_User_Data_128Byte_1[128];
	HwOutputs.Reader_User_Data_128Byte_1[129] := PlcOutputs.Reader_User_Data_128Byte_1[129];
END_FUNCTION
